afC[0  , 0] := 1.00000E+01; afC[0  , 1] := 1.76331E+00;
afC[1  , 0] := 1.99800E+01; afC[1  , 1] := 1.50760E+00;
afC[2  , 0] := 2.99600E+01; afC[2  , 1] := 1.42075E+00;
afC[3  , 0] := 3.99400E+01; afC[3  , 1] := 1.29546E+00;
afC[4  , 0] := 4.99200E+01; afC[4  , 1] := 1.15214E+00;
afC[5  , 0] := 5.99000E+01; afC[5  , 1] := 1.01763E+00;
afC[6  , 0] := 6.98800E+01; afC[6  , 1] := 9.00494E-01;
afC[7  , 0] := 7.98600E+01; afC[7  , 1] := 8.01146E-01;
afC[8  , 0] := 8.98400E+01; afC[8  , 1] := 7.16659E-01;
afC[9  , 0] := 9.98200E+01; afC[9  , 1] := 6.44674E-01;
afC[10 , 0] := 1.09800E+02; afC[10 , 1] := 5.83258E-01;
afC[11 , 0] := 1.19780E+02; afC[11 , 1] := 5.30612E-01;
afC[12 , 0] := 1.29760E+02; afC[12 , 1] := 4.82622E-01;
afC[13 , 0] := 1.39740E+02; afC[13 , 1] := 4.41233E-01;
afC[14 , 0] := 1.49720E+02; afC[14 , 1] := 4.05363E-01;
afC[15 , 0] := 1.59700E+02; afC[15 , 1] := 3.74061E-01;
afC[16 , 0] := 1.69680E+02; afC[16 , 1] := 3.46568E-01;
afC[17 , 0] := 1.79660E+02; afC[17 , 1] := 3.22281E-01;
afC[18 , 0] := 1.89640E+02; afC[18 , 1] := 3.00702E-01;
afC[19 , 0] := 1.99620E+02; afC[19 , 1] := 2.81430E-01;
afC[20 , 0] := 2.09600E+02; afC[20 , 1] := 2.64143E-01;
afC[21 , 0] := 2.19580E+02; afC[21 , 1] := 2.49090E-01;
afC[22 , 0] := 2.29560E+02; afC[22 , 1] := 2.35204E-01;
afC[23 , 0] := 2.39540E+02; afC[23 , 1] := 2.22562E-01;
afC[24 , 0] := 2.49520E+02; afC[24 , 1] := 2.11150E-01;
afC[25 , 0] := 2.59500E+02; afC[25 , 1] := 2.00952E-01;
afC[26 , 0] := 2.69480E+02; afC[26 , 1] := 1.92300E-01;
afC[27 , 0] := 2.79460E+02; afC[27 , 1] := 1.90036E-01;
afC[28 , 0] := 2.89440E+02; afC[28 , 1] := 3.87092E+00;
afC[29 , 0] := 2.99420E+02; afC[29 , 1] := 3.73978E+00;
afC[30 , 0] := 3.09400E+02; afC[30 , 1] := 3.61374E+00;
afC[31 , 0] := 3.19380E+02; afC[31 , 1] := 3.49365E+00;
afC[32 , 0] := 3.29360E+02; afC[32 , 1] := 3.37555E+00;
afC[33 , 0] := 3.39340E+02; afC[33 , 1] := 3.25992E+00;
afC[34 , 0] := 3.49320E+02; afC[34 , 1] := 3.14769E+00;
afC[35 , 0] := 3.59300E+02; afC[35 , 1] := 3.03887E+00;
afC[36 , 0] := 3.69280E+02; afC[36 , 1] := 2.93349E+00;
afC[37 , 0] := 3.79260E+02; afC[37 , 1] := 2.83161E+00;
afC[38 , 0] := 3.89240E+02; afC[38 , 1] := 2.73380E+00;
afC[39 , 0] := 3.99220E+02; afC[39 , 1] := 2.64002E+00;
afC[40 , 0] := 4.09200E+02; afC[40 , 1] := 2.55009E+00;
afC[41 , 0] := 4.19180E+02; afC[41 , 1] := 2.46405E+00;
afC[42 , 0] := 4.29160E+02; afC[42 , 1] := 2.38175E+00;
afC[43 , 0] := 4.39140E+02; afC[43 , 1] := 2.30302E+00;
afC[44 , 0] := 4.49120E+02; afC[44 , 1] := 2.22778E+00;
afC[45 , 0] := 4.59100E+02; afC[45 , 1] := 2.15582E+00;
afC[46 , 0] := 4.69080E+02; afC[46 , 1] := 2.08703E+00;
afC[47 , 0] := 4.79060E+02; afC[47 , 1] := 2.02128E+00;
afC[48 , 0] := 4.89040E+02; afC[48 , 1] := 1.95840E+00;
afC[49 , 0] := 4.99020E+02; afC[49 , 1] := 1.89825E+00;
afC[50 , 0] := 5.09000E+02; afC[50 , 1] := 1.84069E+00;
afC[51 , 0] := 5.18980E+02; afC[51 , 1] := 1.78566E+00;
afC[52 , 0] := 5.28960E+02; afC[52 , 1] := 1.73294E+00;
afC[53 , 0] := 5.38940E+02; afC[53 , 1] := 1.68243E+00;
afC[54 , 0] := 5.48920E+02; afC[54 , 1] := 1.63403E+00;
afC[55 , 0] := 5.58900E+02; afC[55 , 1] := 1.58768E+00;
afC[56 , 0] := 5.68880E+02; afC[56 , 1] := 1.54316E+00;
afC[57 , 0] := 5.78860E+02; afC[57 , 1] := 1.50047E+00;
afC[58 , 0] := 5.88840E+02; afC[58 , 1] := 1.45950E+00;
afC[59 , 0] := 5.98820E+02; afC[59 , 1] := 1.42015E+00;
afC[60 , 0] := 6.08800E+02; afC[60 , 1] := 1.38232E+00;
afC[61 , 0] := 6.18780E+02; afC[61 , 1] := 1.34605E+00;
afC[62 , 0] := 6.28760E+02; afC[62 , 1] := 1.31107E+00;
afC[63 , 0] := 6.38740E+02; afC[63 , 1] := 1.27742E+00;
afC[64 , 0] := 6.48720E+02; afC[64 , 1] := 1.24507E+00;
afC[65 , 0] := 6.58700E+02; afC[65 , 1] := 1.21392E+00;
afC[66 , 0] := 6.68680E+02; afC[66 , 1] := 1.18394E+00;
afC[67 , 0] := 6.78660E+02; afC[67 , 1] := 1.15506E+00;
afC[68 , 0] := 6.88640E+02; afC[68 , 1] := 1.12719E+00;
afC[69 , 0] := 6.98620E+02; afC[69 , 1] := 1.10028E+00;
afC[70 , 0] := 7.08600E+02; afC[70 , 1] := 1.07436E+00;
afC[71 , 0] := 7.18580E+02; afC[71 , 1] := 1.04930E+00;
afC[72 , 0] := 7.28560E+02; afC[72 , 1] := 1.02513E+00;
afC[73 , 0] := 7.38540E+02; afC[73 , 1] := 1.00175E+00;
afC[74 , 0] := 7.48520E+02; afC[74 , 1] := 9.79159E-01;
afC[75 , 0] := 7.58500E+02; afC[75 , 1] := 9.57327E-01;
afC[76 , 0] := 7.68480E+02; afC[76 , 1] := 9.36210E-01;
afC[77 , 0] := 7.78460E+02; afC[77 , 1] := 9.15783E-01;
afC[78 , 0] := 7.88440E+02; afC[78 , 1] := 8.96007E-01;
afC[79 , 0] := 7.98420E+02; afC[79 , 1] := 8.76865E-01;
afC[80 , 0] := 8.08400E+02; afC[80 , 1] := 8.58327E-01;
afC[81 , 0] := 8.18380E+02; afC[81 , 1] := 8.40363E-01;
afC[82 , 0] := 8.28360E+02; afC[82 , 1] := 8.22948E-01;
afC[83 , 0] := 8.38340E+02; afC[83 , 1] := 8.06071E-01;
afC[84 , 0] := 8.48320E+02; afC[84 , 1] := 7.89702E-01;
afC[85 , 0] := 8.58300E+02; afC[85 , 1] := 7.73825E-01;
afC[86 , 0] := 8.68280E+02; afC[86 , 1] := 7.58419E-01;
afC[87 , 0] := 8.78260E+02; afC[87 , 1] := 7.43465E-01;
afC[88 , 0] := 8.88240E+02; afC[88 , 1] := 7.28939E-01;
afC[89 , 0] := 8.98220E+02; afC[89 , 1] := 7.14835E-01;
afC[90 , 0] := 9.08200E+02; afC[90 , 1] := 7.01136E-01;
afC[91 , 0] := 9.18180E+02; afC[91 , 1] := 6.87817E-01;
afC[92 , 0] := 9.28160E+02; afC[92 , 1] := 6.74868E-01;
afC[93 , 0] := 9.38140E+02; afC[93 , 1] := 6.62286E-01;
afC[94 , 0] := 9.48120E+02; afC[94 , 1] := 6.50047E-01;
afC[95 , 0] := 9.58100E+02; afC[95 , 1] := 6.38137E-01;
afC[96 , 0] := 9.68080E+02; afC[96 , 1] := 6.26556E-01;
afC[97 , 0] := 9.78060E+02; afC[97 , 1] := 6.15276E-01;
afC[98 , 0] := 9.88040E+02; afC[98 , 1] := 6.04299E-01;
afC[99 , 0] := 9.98020E+02; afC[99 , 1] := 5.93605E-01;
afC[100, 0] := 1.00800E+03; afC[100, 1] := 5.83149E-01;
afC[101, 0] := 1.01798E+03; afC[101, 1] := 5.72944E-01;
afC[102, 0] := 1.02796E+03; afC[102, 1] := 5.63003E-01;
afC[103, 0] := 1.03794E+03; afC[103, 1] := 5.53309E-01;
afC[104, 0] := 1.04792E+03; afC[104, 1] := 5.43857E-01;
afC[105, 0] := 1.05790E+03; afC[105, 1] := 5.34649E-01;
afC[106, 0] := 1.06788E+03; afC[106, 1] := 5.25672E-01;
afC[107, 0] := 1.07786E+03; afC[107, 1] := 5.16911E-01;
afC[108, 0] := 1.08784E+03; afC[108, 1] := 5.08374E-01;
afC[109, 0] := 1.09782E+03; afC[109, 1] := 5.00040E-01;
afC[110, 0] := 1.10780E+03; afC[110, 1] := 4.91914E-01;
afC[111, 0] := 1.11778E+03; afC[111, 1] := 4.83987E-01;
afC[112, 0] := 1.12776E+03; afC[112, 1] := 4.76243E-01;
afC[113, 0] := 1.13774E+03; afC[113, 1] := 4.68582E-01;
afC[114, 0] := 1.14772E+03; afC[114, 1] := 4.60764E-01;
afC[115, 0] := 1.15770E+03; afC[115, 1] := 4.53142E-01;
afC[116, 0] := 1.16768E+03; afC[116, 1] := 4.45714E-01;
afC[117, 0] := 1.17766E+03; afC[117, 1] := 4.38467E-01;
afC[118, 0] := 1.18764E+03; afC[118, 1] := 4.31397E-01;
afC[119, 0] := 1.19762E+03; afC[119, 1] := 4.24497E-01;
afC[120, 0] := 1.20760E+03; afC[120, 1] := 4.17760E-01;
afC[121, 0] := 1.21758E+03; afC[121, 1] := 4.11188E-01;
afC[122, 0] := 1.22756E+03; afC[122, 1] := 4.04779E-01;
afC[123, 0] := 1.23754E+03; afC[123, 1] := 3.98516E-01;
afC[124, 0] := 1.24752E+03; afC[124, 1] := 3.92394E-01;
afC[125, 0] := 1.25750E+03; afC[125, 1] := 3.86415E-01;
afC[126, 0] := 1.26748E+03; afC[126, 1] := 3.80576E-01;
afC[127, 0] := 1.27746E+03; afC[127, 1] := 3.74871E-01;
afC[128, 0] := 1.28744E+03; afC[128, 1] := 3.69290E-01;
afC[129, 0] := 1.29742E+03; afC[129, 1] := 3.63839E-01;
afC[130, 0] := 1.30740E+03; afC[130, 1] := 3.58513E-01;
afC[131, 0] := 1.31738E+03; afC[131, 1] := 3.53298E-01;
afC[132, 0] := 1.32736E+03; afC[132, 1] := 3.48197E-01;
afC[133, 0] := 1.33734E+03; afC[133, 1] := 3.43209E-01;
afC[134, 0] := 1.34732E+03; afC[134, 1] := 3.38328E-01;
afC[135, 0] := 1.35730E+03; afC[135, 1] := 3.33549E-01;
afC[136, 0] := 1.36728E+03; afC[136, 1] := 3.28877E-01;
afC[137, 0] := 1.37726E+03; afC[137, 1] := 3.24305E-01;
afC[138, 0] := 1.38724E+03; afC[138, 1] := 3.19827E-01;
afC[139, 0] := 1.39722E+03; afC[139, 1] := 3.15438E-01;
afC[140, 0] := 1.40720E+03; afC[140, 1] := 3.11142E-01;
afC[141, 0] := 1.41718E+03; afC[141, 1] := 3.06937E-01;
afC[142, 0] := 1.42716E+03; afC[142, 1] := 3.02821E-01;
afC[143, 0] := 1.43714E+03; afC[143, 1] := 2.98780E-01;
afC[144, 0] := 1.44712E+03; afC[144, 1] := 2.94825E-01;
afC[145, 0] := 1.45710E+03; afC[145, 1] := 2.90951E-01;
afC[146, 0] := 1.46708E+03; afC[146, 1] := 2.87151E-01;
afC[147, 0] := 1.47706E+03; afC[147, 1] := 2.83423E-01;
afC[148, 0] := 1.48704E+03; afC[148, 1] := 2.79767E-01;
afC[149, 0] := 1.49702E+03; afC[149, 1] := 2.76186E-01;
afC[150, 0] := 1.50700E+03; afC[150, 1] := 2.72675E-01;
afC[151, 0] := 1.51698E+03; afC[151, 1] := 2.69230E-01;
afC[152, 0] := 1.52696E+03; afC[152, 1] := 2.65852E-01;
afC[153, 0] := 1.53694E+03; afC[153, 1] := 2.62539E-01;
afC[154, 0] := 1.54692E+03; afC[154, 1] := 2.59288E-01;
afC[155, 0] := 1.55690E+03; afC[155, 1] := 2.56095E-01;
afC[156, 0] := 1.56688E+03; afC[156, 1] := 2.52961E-01;
afC[157, 0] := 1.57686E+03; afC[157, 1] := 2.49883E-01;
afC[158, 0] := 1.58684E+03; afC[158, 1] := 2.46866E-01;
afC[159, 0] := 1.59682E+03; afC[159, 1] := 2.43905E-01;
afC[160, 0] := 1.60680E+03; afC[160, 1] := 2.40998E-01;
afC[161, 0] := 1.61678E+03; afC[161, 1] := 2.38138E-01;
afC[162, 0] := 1.62676E+03; afC[162, 1] := 2.35331E-01;
afC[163, 0] := 1.63674E+03; afC[163, 1] := 2.32580E-01;
afC[164, 0] := 1.64672E+03; afC[164, 1] := 2.29872E-01;
afC[165, 0] := 1.65670E+03; afC[165, 1] := 2.27208E-01;
afC[166, 0] := 1.66668E+03; afC[166, 1] := 2.24594E-01;
afC[167, 0] := 1.67666E+03; afC[167, 1] := 2.22028E-01;
afC[168, 0] := 1.68664E+03; afC[168, 1] := 2.19509E-01;
afC[169, 0] := 1.69662E+03; afC[169, 1] := 2.17030E-01;
afC[170, 0] := 1.70660E+03; afC[170, 1] := 2.14591E-01;
afC[171, 0] := 1.71658E+03; afC[171, 1] := 2.12193E-01;
afC[172, 0] := 1.72656E+03; afC[172, 1] := 2.09837E-01;
afC[173, 0] := 1.73654E+03; afC[173, 1] := 2.07521E-01;
afC[174, 0] := 1.74652E+03; afC[174, 1] := 2.05243E-01;
afC[175, 0] := 1.75650E+03; afC[175, 1] := 2.03000E-01;
afC[176, 0] := 1.76648E+03; afC[176, 1] := 2.00797E-01;
afC[177, 0] := 1.77646E+03; afC[177, 1] := 1.98631E-01;
afC[178, 0] := 1.78644E+03; afC[178, 1] := 1.96498E-01;
afC[179, 0] := 1.79642E+03; afC[179, 1] := 1.94401E-01;
afC[180, 0] := 1.80640E+03; afC[180, 1] := 1.92342E-01;
afC[181, 0] := 1.81638E+03; afC[181, 1] := 1.90313E-01;
afC[182, 0] := 1.82636E+03; afC[182, 1] := 1.88314E-01;
afC[183, 0] := 1.83634E+03; afC[183, 1] := 1.86346E-01;
afC[184, 0] := 1.84632E+03; afC[184, 1] := 1.84410E-01;
afC[185, 0] := 1.85630E+03; afC[185, 1] := 1.82505E-01;
afC[186, 0] := 1.86628E+03; afC[186, 1] := 1.80630E-01;
afC[187, 0] := 1.87626E+03; afC[187, 1] := 1.78786E-01;
afC[188, 0] := 1.88624E+03; afC[188, 1] := 1.76971E-01;
afC[189, 0] := 1.89622E+03; afC[189, 1] := 1.75181E-01;
afC[190, 0] := 1.90620E+03; afC[190, 1] := 1.73419E-01;
afC[191, 0] := 1.91618E+03; afC[191, 1] := 1.71686E-01;
afC[192, 0] := 1.92616E+03; afC[192, 1] := 1.69979E-01;
afC[193, 0] := 1.93614E+03; afC[193, 1] := 1.68292E-01;
afC[194, 0] := 1.94612E+03; afC[194, 1] := 1.66631E-01;
afC[195, 0] := 1.95610E+03; afC[195, 1] := 1.64998E-01;
afC[196, 0] := 1.96608E+03; afC[196, 1] := 1.63390E-01;
afC[197, 0] := 1.97606E+03; afC[197, 1] := 1.61805E-01;
afC[198, 0] := 1.98604E+03; afC[198, 1] := 1.60243E-01;
afC[199, 0] := 1.99602E+03; afC[199, 1] := 1.58705E-01;
afC[200, 0] := 2.00600E+03; afC[200, 1] := 1.57187E-01;
afC[201, 0] := 2.01598E+03; afC[201, 1] := 1.55689E-01;
afC[202, 0] := 2.02596E+03; afC[202, 1] := 1.54215E-01;
afC[203, 0] := 2.03594E+03; afC[203, 1] := 1.52766E-01;
afC[204, 0] := 2.04592E+03; afC[204, 1] := 1.51337E-01;
afC[205, 0] := 2.05590E+03; afC[205, 1] := 1.49926E-01;
afC[206, 0] := 2.06588E+03; afC[206, 1] := 1.48534E-01;
afC[207, 0] := 2.07586E+03; afC[207, 1] := 1.47161E-01;
afC[208, 0] := 2.08584E+03; afC[208, 1] := 1.45807E-01;
afC[209, 0] := 2.09582E+03; afC[209, 1] := 1.44474E-01;
afC[210, 0] := 2.10580E+03; afC[210, 1] := 1.43160E-01;
afC[211, 0] := 2.11578E+03; afC[211, 1] := 1.41862E-01;
afC[212, 0] := 2.12576E+03; afC[212, 1] := 1.40583E-01;
afC[213, 0] := 2.13574E+03; afC[213, 1] := 1.39320E-01;
afC[214, 0] := 2.14572E+03; afC[214, 1] := 1.38074E-01;
afC[215, 0] := 2.15570E+03; afC[215, 1] := 1.36845E-01;
afC[216, 0] := 2.16568E+03; afC[216, 1] := 1.35632E-01;
afC[217, 0] := 2.17566E+03; afC[217, 1] := 1.34436E-01;
afC[218, 0] := 2.18564E+03; afC[218, 1] := 1.33256E-01;
afC[219, 0] := 2.19562E+03; afC[219, 1] := 1.32091E-01;
afC[220, 0] := 2.20560E+03; afC[220, 1] := 1.30943E-01;
afC[221, 0] := 2.21558E+03; afC[221, 1] := 1.29809E-01;
afC[222, 0] := 2.22556E+03; afC[222, 1] := 1.28692E-01;
afC[223, 0] := 2.23554E+03; afC[223, 1] := 1.27588E-01;
afC[224, 0] := 2.24552E+03; afC[224, 1] := 1.26496E-01;
afC[225, 0] := 2.25550E+03; afC[225, 1] := 1.25418E-01;
afC[226, 0] := 2.26548E+03; afC[226, 1] := 1.24360E-01;
afC[227, 0] := 2.27546E+03; afC[227, 1] := 1.23315E-01;
afC[228, 0] := 2.28544E+03; afC[228, 1] := 1.22280E-01;
afC[229, 0] := 2.29542E+03; afC[229, 1] := 1.21256E-01;
afC[230, 0] := 2.30540E+03; afC[230, 1] := 1.20245E-01;
afC[231, 0] := 2.31538E+03; afC[231, 1] := 1.19249E-01;
afC[232, 0] := 2.32536E+03; afC[232, 1] := 1.18265E-01;
afC[233, 0] := 2.33534E+03; afC[233, 1] := 1.17296E-01;
afC[234, 0] := 2.34532E+03; afC[234, 1] := 1.16340E-01;
afC[235, 0] := 2.35530E+03; afC[235, 1] := 1.15391E-01;
afC[236, 0] := 2.36528E+03; afC[236, 1] := 1.14452E-01;
afC[237, 0] := 2.37526E+03; afC[237, 1] := 1.13527E-01;
afC[238, 0] := 2.38524E+03; afC[238, 1] := 1.12614E-01;
afC[239, 0] := 2.39522E+03; afC[239, 1] := 1.11713E-01;
afC[240, 0] := 2.40520E+03; afC[240, 1] := 1.10822E-01;
afC[241, 0] := 2.41518E+03; afC[241, 1] := 1.09942E-01;
afC[242, 0] := 2.42516E+03; afC[242, 1] := 1.09073E-01;
afC[243, 0] := 2.43514E+03; afC[243, 1] := 1.08214E-01;
afC[244, 0] := 2.44512E+03; afC[244, 1] := 1.07365E-01;
afC[245, 0] := 2.45510E+03; afC[245, 1] := 1.06527E-01;
afC[246, 0] := 2.46508E+03; afC[246, 1] := 1.05698E-01;
afC[247, 0] := 2.47506E+03; afC[247, 1] := 1.04879E-01;
afC[248, 0] := 2.48504E+03; afC[248, 1] := 1.04071E-01;
afC[249, 0] := 2.49502E+03; afC[249, 1] := 1.03272E-01;
afC[250, 0] := 2.50500E+03; afC[250, 1] := 1.02482E-01;
afC[251, 0] := 2.51498E+03; afC[251, 1] := 1.01702E-01;
afC[252, 0] := 2.52496E+03; afC[252, 1] := 1.00928E-01;
afC[253, 0] := 2.53494E+03; afC[253, 1] := 1.00163E-01;
afC[254, 0] := 2.54492E+03; afC[254, 1] := 9.94062E-02;
afC[255, 0] := 2.55490E+03; afC[255, 1] := 9.86599E-02;
afC[256, 0] := 2.56488E+03; afC[256, 1] := 9.79221E-02;
afC[257, 0] := 2.57486E+03; afC[257, 1] := 9.71926E-02;
afC[258, 0] := 2.58484E+03; afC[258, 1] := 9.64715E-02;
afC[259, 0] := 2.59482E+03; afC[259, 1] := 9.57584E-02;
afC[260, 0] := 2.60480E+03; afC[260, 1] := 9.50532E-02;
afC[261, 0] := 2.61478E+03; afC[261, 1] := 9.43559E-02;
afC[262, 0] := 2.62476E+03; afC[262, 1] := 9.36664E-02;
afC[263, 0] := 2.63474E+03; afC[263, 1] := 9.29846E-02;
afC[264, 0] := 2.64472E+03; afC[264, 1] := 9.23104E-02;
afC[265, 0] := 2.65470E+03; afC[265, 1] := 9.16432E-02;
afC[266, 0] := 2.66468E+03; afC[266, 1] := 9.09833E-02;
afC[267, 0] := 2.67466E+03; afC[267, 1] := 9.03306E-02;
afC[268, 0] := 2.68464E+03; afC[268, 1] := 8.96849E-02;
afC[269, 0] := 2.69462E+03; afC[269, 1] := 8.90462E-02;
afC[270, 0] := 2.70460E+03; afC[270, 1] := 8.84147E-02;
afC[271, 0] := 2.71458E+03; afC[271, 1] := 8.77902E-02;
afC[272, 0] := 2.72456E+03; afC[272, 1] := 8.71723E-02;
afC[273, 0] := 2.73454E+03; afC[273, 1] := 8.65608E-02;
afC[274, 0] := 2.74452E+03; afC[274, 1] := 8.59557E-02;
afC[275, 0] := 2.75450E+03; afC[275, 1] := 8.53569E-02;
afC[276, 0] := 2.76448E+03; afC[276, 1] := 8.47644E-02;
afC[277, 0] := 2.77446E+03; afC[277, 1] := 8.41781E-02;
afC[278, 0] := 2.78444E+03; afC[278, 1] := 8.35981E-02;
afC[279, 0] := 2.79442E+03; afC[279, 1] := 8.30244E-02;
afC[280, 0] := 2.80440E+03; afC[280, 1] := 8.24567E-02;
afC[281, 0] := 2.81438E+03; afC[281, 1] := 8.18946E-02;
afC[282, 0] := 2.82436E+03; afC[282, 1] := 8.13382E-02;
afC[283, 0] := 2.83434E+03; afC[283, 1] := 8.07874E-02;
afC[284, 0] := 2.84432E+03; afC[284, 1] := 8.02425E-02;
afC[285, 0] := 2.85430E+03; afC[285, 1] := 7.97031E-02;
afC[286, 0] := 2.86428E+03; afC[286, 1] := 7.91692E-02;
afC[287, 0] := 2.87426E+03; afC[287, 1] := 7.86410E-02;
afC[288, 0] := 2.88424E+03; afC[288, 1] := 7.81182E-02;
afC[289, 0] := 2.89422E+03; afC[289, 1] := 7.76006E-02;
afC[290, 0] := 2.90420E+03; afC[290, 1] := 7.70877E-02;
afC[291, 0] := 2.91418E+03; afC[291, 1] := 7.65800E-02;
afC[292, 0] := 2.92416E+03; afC[292, 1] := 7.60774E-02;
afC[293, 0] := 2.93414E+03; afC[293, 1] := 7.55801E-02;
afC[294, 0] := 2.94412E+03; afC[294, 1] := 7.50877E-02;
afC[295, 0] := 2.95410E+03; afC[295, 1] := 7.46001E-02;
afC[296, 0] := 2.96408E+03; afC[296, 1] := 7.41172E-02;
afC[297, 0] := 2.97406E+03; afC[297, 1] := 7.36390E-02;
afC[298, 0] := 2.98404E+03; afC[298, 1] := 7.31616E-02;
afC[299, 0] := 2.99402E+03; afC[299, 1] := 7.26796E-02;
afC[300, 0] := 3.00400E+03; afC[300, 1] := 7.22023E-02;
afC[301, 0] := 3.01398E+03; afC[301, 1] := 7.17227E-02;
afC[302, 0] := 3.02396E+03; afC[302, 1] := 7.12320E-02;
afC[303, 0] := 3.03394E+03; afC[303, 1] := 7.07462E-02;
afC[304, 0] := 3.04392E+03; afC[304, 1] := 7.02654E-02;
afC[305, 0] := 3.05390E+03; afC[305, 1] := 6.97897E-02;
afC[306, 0] := 3.06388E+03; afC[306, 1] := 6.93187E-02;
afC[307, 0] := 3.07386E+03; afC[307, 1] := 6.88524E-02;
afC[308, 0] := 3.08384E+03; afC[308, 1] := 6.83906E-02;
afC[309, 0] := 3.09382E+03; afC[309, 1] := 6.79334E-02;
afC[310, 0] := 3.10380E+03; afC[310, 1] := 6.74808E-02;
afC[311, 0] := 3.11378E+03; afC[311, 1] := 6.70329E-02;
afC[312, 0] := 3.12376E+03; afC[312, 1] := 6.65895E-02;
afC[313, 0] := 3.13374E+03; afC[313, 1] := 6.61503E-02;
afC[314, 0] := 3.14372E+03; afC[314, 1] := 6.57151E-02;
afC[315, 0] := 3.15370E+03; afC[315, 1] := 6.52841E-02;
afC[316, 0] := 3.16368E+03; afC[316, 1] := 6.48572E-02;
afC[317, 0] := 3.17366E+03; afC[317, 1] := 6.44346E-02;
afC[318, 0] := 3.18364E+03; afC[318, 1] := 6.40161E-02;
afC[319, 0] := 3.19362E+03; afC[319, 1] := 6.36016E-02;
afC[320, 0] := 3.20360E+03; afC[320, 1] := 6.31910E-02;
afC[321, 0] := 3.21358E+03; afC[321, 1] := 6.27843E-02;
afC[322, 0] := 3.22356E+03; afC[322, 1] := 6.23815E-02;
afC[323, 0] := 3.23354E+03; afC[323, 1] := 6.19824E-02;
afC[324, 0] := 3.24352E+03; afC[324, 1] := 6.15871E-02;
afC[325, 0] := 3.25350E+03; afC[325, 1] := 6.11954E-02;
afC[326, 0] := 3.26348E+03; afC[326, 1] := 6.08075E-02;
afC[327, 0] := 3.27346E+03; afC[327, 1] := 6.04235E-02;
afC[328, 0] := 3.28344E+03; afC[328, 1] := 6.00430E-02;
afC[329, 0] := 3.29342E+03; afC[329, 1] := 5.96661E-02;
afC[330, 0] := 3.30340E+03; afC[330, 1] := 5.92926E-02;
afC[331, 0] := 3.31338E+03; afC[331, 1] := 5.89225E-02;
afC[332, 0] := 3.32336E+03; afC[332, 1] := 5.85558E-02;
afC[333, 0] := 3.33334E+03; afC[333, 1] := 5.81925E-02;
afC[334, 0] := 3.34332E+03; afC[334, 1] := 5.78325E-02;
afC[335, 0] := 3.35330E+03; afC[335, 1] := 5.74758E-02;
afC[336, 0] := 3.36328E+03; afC[336, 1] := 5.71223E-02;
afC[337, 0] := 3.37326E+03; afC[337, 1] := 5.67720E-02;
afC[338, 0] := 3.38324E+03; afC[338, 1] := 5.64248E-02;
afC[339, 0] := 3.39322E+03; afC[339, 1] := 5.60808E-02;
afC[340, 0] := 3.40320E+03; afC[340, 1] := 5.57402E-02;
afC[341, 0] := 3.41318E+03; afC[341, 1] := 5.54026E-02;
afC[342, 0] := 3.42316E+03; afC[342, 1] := 5.50681E-02;
afC[343, 0] := 3.43314E+03; afC[343, 1] := 5.47363E-02;
afC[344, 0] := 3.44312E+03; afC[344, 1] := 5.44072E-02;
afC[345, 0] := 3.45310E+03; afC[345, 1] := 5.40811E-02;
afC[346, 0] := 3.46308E+03; afC[346, 1] := 5.37580E-02;
afC[347, 0] := 3.47306E+03; afC[347, 1] := 5.34379E-02;
afC[348, 0] := 3.48304E+03; afC[348, 1] := 5.31207E-02;
afC[349, 0] := 3.49302E+03; afC[349, 1] := 5.28062E-02;
afC[350, 0] := 3.50300E+03; afC[350, 1] := 5.24944E-02;
afC[351, 0] := 3.51298E+03; afC[351, 1] := 5.21853E-02;
afC[352, 0] := 3.52296E+03; afC[352, 1] := 5.18788E-02;
afC[353, 0] := 3.53294E+03; afC[353, 1] := 5.15750E-02;
afC[354, 0] := 3.54292E+03; afC[354, 1] := 5.12739E-02;
afC[355, 0] := 3.55290E+03; afC[355, 1] := 5.09753E-02;
afC[356, 0] := 3.56288E+03; afC[356, 1] := 5.06793E-02;
afC[357, 0] := 3.57286E+03; afC[357, 1] := 5.03859E-02;
afC[358, 0] := 3.58284E+03; afC[358, 1] := 5.00951E-02;
afC[359, 0] := 3.59282E+03; afC[359, 1] := 4.98067E-02;
afC[360, 0] := 3.60280E+03; afC[360, 1] := 4.95208E-02;
afC[361, 0] := 3.61278E+03; afC[361, 1] := 4.92373E-02;
afC[362, 0] := 3.62276E+03; afC[362, 1] := 4.89562E-02;
afC[363, 0] := 3.63274E+03; afC[363, 1] := 4.86774E-02;
afC[364, 0] := 3.64272E+03; afC[364, 1] := 4.84011E-02;
afC[365, 0] := 3.65270E+03; afC[365, 1] := 4.81271E-02;
afC[366, 0] := 3.66268E+03; afC[366, 1] := 4.78554E-02;
afC[367, 0] := 3.67266E+03; afC[367, 1] := 4.75859E-02;
afC[368, 0] := 3.68264E+03; afC[368, 1] := 4.73187E-02;
afC[369, 0] := 3.69262E+03; afC[369, 1] := 4.70536E-02;
afC[370, 0] := 3.70260E+03; afC[370, 1] := 4.67908E-02;
afC[371, 0] := 3.71258E+03; afC[371, 1] := 4.65301E-02;
afC[372, 0] := 3.72256E+03; afC[372, 1] := 4.62716E-02;
afC[373, 0] := 3.73254E+03; afC[373, 1] := 4.60152E-02;
afC[374, 0] := 3.74252E+03; afC[374, 1] := 4.57609E-02;
afC[375, 0] := 3.75250E+03; afC[375, 1] := 4.55086E-02;
afC[376, 0] := 3.76248E+03; afC[376, 1] := 4.52583E-02;
afC[377, 0] := 3.77246E+03; afC[377, 1] := 4.50101E-02;
afC[378, 0] := 3.78244E+03; afC[378, 1] := 4.47639E-02;
afC[379, 0] := 3.79242E+03; afC[379, 1] := 4.45196E-02;
afC[380, 0] := 3.80240E+03; afC[380, 1] := 4.42773E-02;
afC[381, 0] := 3.81238E+03; afC[381, 1] := 4.40370E-02;
afC[382, 0] := 3.82236E+03; afC[382, 1] := 4.37986E-02;
afC[383, 0] := 3.83234E+03; afC[383, 1] := 4.35624E-02;
afC[384, 0] := 3.84232E+03; afC[384, 1] := 4.33281E-02;
afC[385, 0] := 3.85230E+03; afC[385, 1] := 4.30957E-02;
afC[386, 0] := 3.86228E+03; afC[386, 1] := 4.28651E-02;
afC[387, 0] := 3.87226E+03; afC[387, 1] := 4.26360E-02;
afC[388, 0] := 3.88224E+03; afC[388, 1] := 4.24087E-02;
afC[389, 0] := 3.89222E+03; afC[389, 1] := 4.21833E-02;
afC[390, 0] := 3.90220E+03; afC[390, 1] := 4.19596E-02;
afC[391, 0] := 3.91218E+03; afC[391, 1] := 4.17376E-02;
afC[392, 0] := 3.92216E+03; afC[392, 1] := 4.15174E-02;
afC[393, 0] := 3.93214E+03; afC[393, 1] := 4.12989E-02;
afC[394, 0] := 3.94212E+03; afC[394, 1] := 4.10822E-02;
afC[395, 0] := 3.95210E+03; afC[395, 1] := 4.08672E-02;
afC[396, 0] := 3.96208E+03; afC[396, 1] := 4.06539E-02;
afC[397, 0] := 3.97206E+03; afC[397, 1] := 4.04422E-02;
afC[398, 0] := 3.98204E+03; afC[398, 1] := 4.02321E-02;
afC[399, 0] := 3.99202E+03; afC[399, 1] := 4.00236E-02;
afC[400, 0] := 4.00200E+03; afC[400, 1] := 3.98167E-02;
afC[401, 0] := 4.01198E+03; afC[401, 1] := 3.96114E-02;
afC[402, 0] := 4.02196E+03; afC[402, 1] := 3.94077E-02;
afC[403, 0] := 4.03194E+03; afC[403, 1] := 3.92055E-02;
afC[404, 0] := 4.04192E+03; afC[404, 1] := 3.90049E-02;
afC[405, 0] := 4.05190E+03; afC[405, 1] := 3.88058E-02;
afC[406, 0] := 4.06188E+03; afC[406, 1] := 3.86082E-02;
afC[407, 0] := 4.07186E+03; afC[407, 1] := 3.84119E-02;
afC[408, 0] := 4.08184E+03; afC[408, 1] := 3.82172E-02;
afC[409, 0] := 4.09182E+03; afC[409, 1] := 3.80239E-02;
afC[410, 0] := 4.10180E+03; afC[410, 1] := 3.78321E-02;
afC[411, 0] := 4.11178E+03; afC[411, 1] := 3.76418E-02;
afC[412, 0] := 4.12176E+03; afC[412, 1] := 3.74530E-02;
afC[413, 0] := 4.13174E+03; afC[413, 1] := 3.72656E-02;
afC[414, 0] := 4.14172E+03; afC[414, 1] := 3.70795E-02;
afC[415, 0] := 4.15170E+03; afC[415, 1] := 3.68947E-02;
afC[416, 0] := 4.16168E+03; afC[416, 1] := 3.67112E-02;
afC[417, 0] := 4.17166E+03; afC[417, 1] := 3.65291E-02;
afC[418, 0] := 4.18164E+03; afC[418, 1] := 3.63483E-02;
afC[419, 0] := 4.19162E+03; afC[419, 1] := 3.61689E-02;
afC[420, 0] := 4.20160E+03; afC[420, 1] := 3.59908E-02;
afC[421, 0] := 4.21158E+03; afC[421, 1] := 3.58141E-02;
afC[422, 0] := 4.22156E+03; afC[422, 1] := 3.56386E-02;
afC[423, 0] := 4.23154E+03; afC[423, 1] := 3.54643E-02;
afC[424, 0] := 4.24152E+03; afC[424, 1] := 3.52914E-02;
afC[425, 0] := 4.25150E+03; afC[425, 1] := 3.51196E-02;
afC[426, 0] := 4.26148E+03; afC[426, 1] := 3.49491E-02;
afC[427, 0] := 4.27146E+03; afC[427, 1] := 3.47798E-02;
afC[428, 0] := 4.28144E+03; afC[428, 1] := 3.46118E-02;
afC[429, 0] := 4.29142E+03; afC[429, 1] := 3.44449E-02;
afC[430, 0] := 4.30140E+03; afC[430, 1] := 3.42793E-02;
afC[431, 0] := 4.31138E+03; afC[431, 1] := 3.41148E-02;
afC[432, 0] := 4.32136E+03; afC[432, 1] := 3.39516E-02;
afC[433, 0] := 4.33134E+03; afC[433, 1] := 3.37896E-02;
afC[434, 0] := 4.34132E+03; afC[434, 1] := 3.36287E-02;
afC[435, 0] := 4.35130E+03; afC[435, 1] := 3.34689E-02;
afC[436, 0] := 4.36128E+03; afC[436, 1] := 3.33099E-02;
afC[437, 0] := 4.37126E+03; afC[437, 1] := 3.31521E-02;
afC[438, 0] := 4.38124E+03; afC[438, 1] := 3.29954E-02;
afC[439, 0] := 4.39122E+03; afC[439, 1] := 3.28397E-02;
afC[440, 0] := 4.40120E+03; afC[440, 1] := 3.26853E-02;
afC[441, 0] := 4.41118E+03; afC[441, 1] := 3.25321E-02;
afC[442, 0] := 4.42116E+03; afC[442, 1] := 3.23799E-02;
afC[443, 0] := 4.43114E+03; afC[443, 1] := 3.22288E-02;
afC[444, 0] := 4.44112E+03; afC[444, 1] := 3.20787E-02;
afC[445, 0] := 4.45110E+03; afC[445, 1] := 3.19297E-02;
afC[446, 0] := 4.46108E+03; afC[446, 1] := 3.17817E-02;
afC[447, 0] := 4.47106E+03; afC[447, 1] := 3.16348E-02;
afC[448, 0] := 4.48104E+03; afC[448, 1] := 3.14888E-02;
afC[449, 0] := 4.49102E+03; afC[449, 1] := 3.13436E-02;
afC[450, 0] := 4.50100E+03; afC[450, 1] := 3.11994E-02;
afC[451, 0] := 4.51098E+03; afC[451, 1] := 3.10561E-02;
afC[452, 0] := 4.52096E+03; afC[452, 1] := 3.09137E-02;
afC[453, 0] := 4.53094E+03; afC[453, 1] := 3.07725E-02;
afC[454, 0] := 4.54092E+03; afC[454, 1] := 3.06325E-02;
afC[455, 0] := 4.55090E+03; afC[455, 1] := 3.04935E-02;
afC[456, 0] := 4.56088E+03; afC[456, 1] := 3.03553E-02;
afC[457, 0] := 4.57086E+03; afC[457, 1] := 3.02181E-02;
afC[458, 0] := 4.58084E+03; afC[458, 1] := 3.00815E-02;
afC[459, 0] := 4.59082E+03; afC[459, 1] := 2.99458E-02;
afC[460, 0] := 4.60080E+03; afC[460, 1] := 2.98109E-02;
afC[461, 0] := 4.61078E+03; afC[461, 1] := 2.96769E-02;
afC[462, 0] := 4.62076E+03; afC[462, 1] := 2.95439E-02;
afC[463, 0] := 4.63074E+03; afC[463, 1] := 2.94120E-02;
afC[464, 0] := 4.64072E+03; afC[464, 1] := 2.92810E-02;
afC[465, 0] := 4.65070E+03; afC[465, 1] := 2.91508E-02;
afC[466, 0] := 4.66068E+03; afC[466, 1] := 2.90215E-02;
afC[467, 0] := 4.67066E+03; afC[467, 1] := 2.88930E-02;
afC[468, 0] := 4.68064E+03; afC[468, 1] := 2.87653E-02;
afC[469, 0] := 4.69062E+03; afC[469, 1] := 2.86384E-02;
afC[470, 0] := 4.70060E+03; afC[470, 1] := 2.85124E-02;
afC[471, 0] := 4.71058E+03; afC[471, 1] := 2.83872E-02;
afC[472, 0] := 4.72056E+03; afC[472, 1] := 2.82628E-02;
afC[473, 0] := 4.73054E+03; afC[473, 1] := 2.81392E-02;
afC[474, 0] := 4.74052E+03; afC[474, 1] := 2.80163E-02;
afC[475, 0] := 4.75050E+03; afC[475, 1] := 2.78943E-02;
afC[476, 0] := 4.76048E+03; afC[476, 1] := 2.77731E-02;
afC[477, 0] := 4.77046E+03; afC[477, 1] := 2.76527E-02;
afC[478, 0] := 4.78044E+03; afC[478, 1] := 2.75330E-02;
afC[479, 0] := 4.79042E+03; afC[479, 1] := 2.74141E-02;
afC[480, 0] := 4.80040E+03; afC[480, 1] := 2.72960E-02;
afC[481, 0] := 4.81038E+03; afC[481, 1] := 2.71785E-02;
afC[482, 0] := 4.82036E+03; afC[482, 1] := 2.70618E-02;
afC[483, 0] := 4.83034E+03; afC[483, 1] := 2.69458E-02;
afC[484, 0] := 4.84032E+03; afC[484, 1] := 2.68305E-02;
afC[485, 0] := 4.85030E+03; afC[485, 1] := 2.67159E-02;
afC[486, 0] := 4.86028E+03; afC[486, 1] := 2.66022E-02;
afC[487, 0] := 4.87026E+03; afC[487, 1] := 2.64892E-02;
afC[488, 0] := 4.88024E+03; afC[488, 1] := 2.63769E-02;
afC[489, 0] := 4.89022E+03; afC[489, 1] := 2.62653E-02;
afC[490, 0] := 4.90020E+03; afC[490, 1] := 2.61545E-02;
afC[491, 0] := 4.91018E+03; afC[491, 1] := 2.60443E-02;
afC[492, 0] := 4.92016E+03; afC[492, 1] := 2.59347E-02;
afC[493, 0] := 4.93014E+03; afC[493, 1] := 2.58259E-02;
afC[494, 0] := 4.94012E+03; afC[494, 1] := 2.57177E-02;
afC[495, 0] := 4.95010E+03; afC[495, 1] := 2.56102E-02;
afC[496, 0] := 4.96008E+03; afC[496, 1] := 2.55034E-02;
afC[497, 0] := 4.97006E+03; afC[497, 1] := 2.53972E-02;
afC[498, 0] := 4.98004E+03; afC[498, 1] := 2.52917E-02;
afC[499, 0] := 4.99002E+03; afC[499, 1] := 2.51869E-02;
afC[500, 0] := 5.00000E+03; afC[500, 1] := 2.50827E-02;
afC[501, 0] := 5.05000E+03; afC[501, 1] := 2.45704E-02;
afC[502, 0] := 5.10000E+03; afC[502, 1] := 2.40730E-02;
afC[503, 0] := 5.15000E+03; afC[503, 1] := 2.35901E-02;
afC[504, 0] := 5.20000E+03; afC[504, 1] := 2.31214E-02;
afC[505, 0] := 5.25000E+03; afC[505, 1] := 2.26673E-02;
afC[506, 0] := 5.30000E+03; afC[506, 1] := 2.22259E-02;
afC[507, 0] := 5.35000E+03; afC[507, 1] := 2.17882E-02;
afC[508, 0] := 5.40000E+03; afC[508, 1] := 2.13564E-02;
afC[509, 0] := 5.45000E+03; afC[509, 1] := 2.09356E-02;
afC[510, 0] := 5.50000E+03; afC[510, 1] := 2.05272E-02;
afC[511, 0] := 5.55000E+03; afC[511, 1] := 2.01302E-02;
afC[512, 0] := 5.60000E+03; afC[512, 1] := 1.97446E-02;
afC[513, 0] := 5.65000E+03; afC[513, 1] := 1.93698E-02;
afC[514, 0] := 5.70000E+03; afC[514, 1] := 1.90048E-02;
afC[515, 0] := 5.75000E+03; afC[515, 1] := 1.86499E-02;
afC[516, 0] := 5.80000E+03; afC[516, 1] := 1.83050E-02;
afC[517, 0] := 5.85000E+03; afC[517, 1] := 1.79691E-02;
afC[518, 0] := 5.90000E+03; afC[518, 1] := 1.76418E-02;
afC[519, 0] := 5.95000E+03; afC[519, 1] := 1.73236E-02;
afC[520, 0] := 6.00000E+03; afC[520, 1] := 1.70139E-02;
afC[521, 0] := 6.05000E+03; afC[521, 1] := 1.67117E-02;
afC[522, 0] := 6.10000E+03; afC[522, 1] := 1.64175E-02;
afC[523, 0] := 6.15000E+03; afC[523, 1] := 1.61304E-02;
afC[524, 0] := 6.20000E+03; afC[524, 1] := 1.58509E-02;
afC[525, 0] := 6.25000E+03; afC[525, 1] := 1.55788E-02;
afC[526, 0] := 6.30000E+03; afC[526, 1] := 1.53136E-02;
afC[527, 0] := 6.35000E+03; afC[527, 1] := 1.50544E-02;
afC[528, 0] := 6.40000E+03; afC[528, 1] := 1.48015E-02;
afC[529, 0] := 6.45000E+03; afC[529, 1] := 1.45549E-02;
afC[530, 0] := 6.50000E+03; afC[530, 1] := 1.43145E-02;
afC[531, 0] := 6.55000E+03; afC[531, 1] := 1.40799E-02;
afC[532, 0] := 6.60000E+03; afC[532, 1] := 1.38506E-02;
afC[533, 0] := 6.65000E+03; afC[533, 1] := 1.36271E-02;
afC[534, 0] := 6.70000E+03; afC[534, 1] := 1.34088E-02;
afC[535, 0] := 6.75000E+03; afC[535, 1] := 1.31956E-02;
afC[536, 0] := 6.80000E+03; afC[536, 1] := 1.29872E-02;
afC[537, 0] := 6.85000E+03; afC[537, 1] := 1.27830E-02;
afC[538, 0] := 6.90000E+03; afC[538, 1] := 1.25837E-02;
afC[539, 0] := 6.95000E+03; afC[539, 1] := 1.23893E-02;
afC[540, 0] := 7.00000E+03; afC[540, 1] := 1.21996E-02;
afC[541, 0] := 7.05000E+03; afC[541, 1] := 1.20137E-02;
afC[542, 0] := 7.10000E+03; afC[542, 1] := 1.18318E-02;
afC[543, 0] := 7.15000E+03; afC[543, 1] := 1.16536E-02;
afC[544, 0] := 7.20000E+03; afC[544, 1] := 1.14797E-02;
afC[545, 0] := 7.25000E+03; afC[545, 1] := 1.13096E-02;
afC[546, 0] := 7.30000E+03; afC[546, 1] := 1.11430E-02;
afC[547, 0] := 7.35000E+03; afC[547, 1] := 1.09806E-02;
afC[548, 0] := 7.40000E+03; afC[548, 1] := 1.08212E-02;
afC[549, 0] := 7.45000E+03; afC[549, 1] := 1.06649E-02;
afC[550, 0] := 7.50000E+03; afC[550, 1] := 1.05119E-02;
afC[551, 0] := 7.55000E+03; afC[551, 1] := 1.03622E-02;
afC[552, 0] := 7.60000E+03; afC[552, 1] := 1.02157E-02;
afC[553, 0] := 7.65000E+03; afC[553, 1] := 1.00723E-02;
afC[554, 0] := 7.70000E+03; afC[554, 1] := 9.93170E-03;
afC[555, 0] := 7.75000E+03; afC[555, 1] := 9.79384E-03;
afC[556, 0] := 7.80000E+03; afC[556, 1] := 9.65888E-03;
afC[557, 0] := 7.85000E+03; afC[557, 1] := 9.52665E-03;
afC[558, 0] := 7.90000E+03; afC[558, 1] := 9.39708E-03;
afC[559, 0] := 7.95000E+03; afC[559, 1] := 9.27001E-03;
afC[560, 0] := 8.00000E+03; afC[560, 1] := 9.14543E-03;
afC[561, 0] := 8.05000E+03; afC[561, 1] := 9.02332E-03;
afC[562, 0] := 8.10000E+03; afC[562, 1] := 8.90356E-03;
afC[563, 0] := 8.15000E+03; afC[563, 1] := 8.78611E-03;
afC[564, 0] := 8.20000E+03; afC[564, 1] := 8.67093E-03;
afC[565, 0] := 8.25000E+03; afC[565, 1] := 8.55793E-03;
afC[566, 0] := 8.30000E+03; afC[566, 1] := 8.44705E-03;
afC[567, 0] := 8.35000E+03; afC[567, 1] := 8.33832E-03;
afC[568, 0] := 8.40000E+03; afC[568, 1] := 8.23162E-03;
afC[569, 0] := 8.45000E+03; afC[569, 1] := 8.12686E-03;
afC[570, 0] := 8.50000E+03; afC[570, 1] := 8.02406E-03;
afC[571, 0] := 8.55000E+03; afC[571, 1] := 7.92318E-03;
afC[572, 0] := 8.60000E+03; afC[572, 1] := 7.82412E-03;
afC[573, 0] := 8.65000E+03; afC[573, 1] := 7.72686E-03;
afC[574, 0] := 8.70000E+03; afC[574, 1] := 7.63138E-03;
afC[575, 0] := 8.75000E+03; afC[575, 1] := 7.53760E-03;
afC[576, 0] := 8.80000E+03; afC[576, 1] := 7.44546E-03;
afC[577, 0] := 8.85000E+03; afC[577, 1] := 7.35477E-03;
afC[578, 0] := 8.90000E+03; afC[578, 1] := 7.26558E-03;
afC[579, 0] := 8.95000E+03; afC[579, 1] := 7.17504E-03;
afC[580, 0] := 9.00000E+03; afC[580, 1] := 7.08565E-03;
afC[581, 0] := 9.05000E+03; afC[581, 1] := 6.99789E-03;
afC[582, 0] := 9.10000E+03; afC[582, 1] := 6.91169E-03;
afC[583, 0] := 9.15000E+03; afC[583, 1] := 6.82703E-03;
afC[584, 0] := 9.20000E+03; afC[584, 1] := 6.74383E-03;
afC[585, 0] := 9.25000E+03; afC[585, 1] := 6.66206E-03;
afC[586, 0] := 9.30000E+03; afC[586, 1] := 6.58175E-03;
afC[587, 0] := 9.35000E+03; afC[587, 1] := 6.50283E-03;
afC[588, 0] := 9.40000E+03; afC[588, 1] := 6.42530E-03;
afC[589, 0] := 9.45000E+03; afC[589, 1] := 6.34910E-03;
afC[590, 0] := 9.50000E+03; afC[590, 1] := 6.27417E-03;
afC[591, 0] := 9.55000E+03; afC[591, 1] := 6.20050E-03;
afC[592, 0] := 9.60000E+03; afC[592, 1] := 6.12807E-03;
afC[593, 0] := 9.65000E+03; afC[593, 1] := 6.05686E-03;
afC[594, 0] := 9.70000E+03; afC[594, 1] := 5.98686E-03;
afC[595, 0] := 9.75000E+03; afC[595, 1] := 5.91802E-03;
afC[596, 0] := 9.80000E+03; afC[596, 1] := 5.85029E-03;
afC[597, 0] := 9.85000E+03; afC[597, 1] := 5.78369E-03;
afC[598, 0] := 9.90000E+03; afC[598, 1] := 5.71821E-03;
afC[599, 0] := 9.95000E+03; afC[599, 1] := 5.65379E-03;
afC[600, 0] := 1.00000E+04; afC[600, 1] := 5.59040E-03;
afC[601, 0] := 1.00500E+04; afC[601, 1] := 5.52802E-03;
afC[602, 0] := 1.01000E+04; afC[602, 1] := 5.46662E-03;
afC[603, 0] := 1.01500E+04; afC[603, 1] := 5.40620E-03;
afC[604, 0] := 1.02000E+04; afC[604, 1] := 5.34677E-03;
afC[605, 0] := 1.02500E+04; afC[605, 1] := 5.28829E-03;
afC[606, 0] := 1.03000E+04; afC[606, 1] := 5.23074E-03;
afC[607, 0] := 1.03500E+04; afC[607, 1] := 5.17409E-03;
afC[608, 0] := 1.04000E+04; afC[608, 1] := 5.11828E-03;
afC[609, 0] := 1.04500E+04; afC[609, 1] := 5.06334E-03;
afC[610, 0] := 1.05000E+04; afC[610, 1] := 5.00927E-03;
afC[611, 0] := 1.05500E+04; afC[611, 1] := 4.95603E-03;
afC[612, 0] := 1.06000E+04; afC[612, 1] := 4.90356E-03;
afC[613, 0] := 1.06500E+04; afC[613, 1] := 4.85190E-03;
afC[614, 0] := 1.07000E+04; afC[614, 1] := 4.80104E-03;
afC[615, 0] := 1.07500E+04; afC[615, 1] := 4.75096E-03;
afC[616, 0] := 1.08000E+04; afC[616, 1] := 4.70163E-03;
afC[617, 0] := 1.08500E+04; afC[617, 1] := 4.65305E-03;
afC[618, 0] := 1.09000E+04; afC[618, 1] := 4.60518E-03;
afC[619, 0] := 1.09500E+04; afC[619, 1] := 4.55801E-03;
afC[620, 0] := 1.10000E+04; afC[620, 1] := 4.51154E-03;
afC[621, 0] := 1.10500E+04; afC[621, 1] := 4.46577E-03;
afC[622, 0] := 1.11000E+04; afC[622, 1] := 4.42065E-03;
afC[623, 0] := 1.11500E+04; afC[623, 1] := 4.37614E-03;
afC[624, 0] := 1.12000E+04; afC[624, 1] := 4.33228E-03;
afC[625, 0] := 1.12500E+04; afC[625, 1] := 4.28910E-03;
afC[626, 0] := 1.13000E+04; afC[626, 1] := 4.24655E-03;
afC[627, 0] := 1.13500E+04; afC[627, 1] := 4.20459E-03;
afC[628, 0] := 1.14000E+04; afC[628, 1] := 4.16323E-03;
afC[629, 0] := 1.14500E+04; afC[629, 1] := 4.12243E-03;
afC[630, 0] := 1.15000E+04; afC[630, 1] := 4.08220E-03;
afC[631, 0] := 1.15500E+04; afC[631, 1] := 4.04253E-03;
afC[632, 0] := 1.16000E+04; afC[632, 1] := 4.00345E-03;
afC[633, 0] := 1.16500E+04; afC[633, 1] := 3.96490E-03;
afC[634, 0] := 1.17000E+04; afC[634, 1] := 3.92690E-03;
afC[635, 0] := 1.17500E+04; afC[635, 1] := 3.88942E-03;
afC[636, 0] := 1.18000E+04; afC[636, 1] := 3.85244E-03;
afC[637, 0] := 1.18500E+04; afC[637, 1] := 3.81597E-03;
afC[638, 0] := 1.19000E+04; afC[638, 1] := 3.77999E-03;
afC[639, 0] := 1.19500E+04; afC[639, 1] := 3.74450E-03;
afC[640, 0] := 1.20000E+04; afC[640, 1] := 3.70948E-03;
afC[641, 0] := 1.20500E+04; afC[641, 1] := 3.67496E-03;
afC[642, 0] := 1.21000E+04; afC[642, 1] := 3.64090E-03;
afC[643, 0] := 1.21500E+04; afC[643, 1] := 3.60729E-03;
afC[644, 0] := 1.22000E+04; afC[644, 1] := 3.57412E-03;
afC[645, 0] := 1.22500E+04; afC[645, 1] := 3.54139E-03;
afC[646, 0] := 1.23000E+04; afC[646, 1] := 3.50906E-03;
afC[647, 0] := 1.23500E+04; afC[647, 1] := 3.47716E-03;
afC[648, 0] := 1.24000E+04; afC[648, 1] := 3.44569E-03;
afC[649, 0] := 1.24500E+04; afC[649, 1] := 3.41464E-03;
afC[650, 0] := 1.25000E+04; afC[650, 1] := 3.38399E-03;
afC[651, 0] := 1.25500E+04; afC[651, 1] := 3.35374E-03;
afC[652, 0] := 1.26000E+04; afC[652, 1] := 3.32387E-03;
afC[653, 0] := 1.26500E+04; afC[653, 1] := 3.29440E-03;
afC[654, 0] := 1.27000E+04; afC[654, 1] := 3.26532E-03;
afC[655, 0] := 1.27500E+04; afC[655, 1] := 3.23660E-03;
afC[656, 0] := 1.28000E+04; afC[656, 1] := 3.20823E-03;
afC[657, 0] := 1.28500E+04; afC[657, 1] := 3.18023E-03;
afC[658, 0] := 1.29000E+04; afC[658, 1] := 3.15255E-03;
afC[659, 0] := 1.29500E+04; afC[659, 1] := 3.12521E-03;
afC[660, 0] := 1.30000E+04; afC[660, 1] := 3.09821E-03;
afC[661, 0] := 1.30500E+04; afC[661, 1] := 3.07156E-03;
afC[662, 0] := 1.31000E+04; afC[662, 1] := 3.04524E-03;
afC[663, 0] := 1.31500E+04; afC[663, 1] := 3.01926E-03;
afC[664, 0] := 1.32000E+04; afC[664, 1] := 2.99362E-03;
afC[665, 0] := 1.32500E+04; afC[665, 1] := 2.96829E-03;
afC[666, 0] := 1.33000E+04; afC[666, 1] := 2.94325E-03;
afC[667, 0] := 1.33500E+04; afC[667, 1] := 2.91850E-03;
afC[668, 0] := 1.34000E+04; afC[668, 1] := 2.89405E-03;
afC[669, 0] := 1.34500E+04; afC[669, 1] := 2.86991E-03;
afC[670, 0] := 1.35000E+04; afC[670, 1] := 2.84607E-03;
afC[671, 0] := 1.35500E+04; afC[671, 1] := 2.82250E-03;
afC[672, 0] := 1.36000E+04; afC[672, 1] := 2.79922E-03;
afC[673, 0] := 1.36500E+04; afC[673, 1] := 2.77621E-03;
afC[674, 0] := 1.37000E+04; afC[674, 1] := 2.75344E-03;
afC[675, 0] := 1.37500E+04; afC[675, 1] := 2.73094E-03;
afC[676, 0] := 1.38000E+04; afC[676, 1] := 2.70870E-03;
afC[677, 0] := 1.38500E+04; afC[677, 1] := 2.68678E-03;
afC[678, 0] := 1.39000E+04; afC[678, 1] := 2.66511E-03;
afC[679, 0] := 1.39500E+04; afC[679, 1] := 2.64369E-03;
afC[680, 0] := 1.40000E+04; afC[680, 1] := 2.62251E-03;
afC[681, 0] := 1.40500E+04; afC[681, 1] := 2.60157E-03;
afC[682, 0] := 1.41000E+04; afC[682, 1] := 2.58086E-03;
afC[683, 0] := 1.41500E+04; afC[683, 1] := 2.56037E-03;
afC[684, 0] := 1.42000E+04; afC[684, 1] := 2.54011E-03;
afC[685, 0] := 1.42500E+04; afC[685, 1] := 2.52011E-03;
afC[686, 0] := 1.43000E+04; afC[686, 1] := 2.50035E-03;
afC[687, 0] := 1.43500E+04; afC[687, 1] := 2.48082E-03;
afC[688, 0] := 1.44000E+04; afC[688, 1] := 2.46147E-03;
afC[689, 0] := 1.44500E+04; afC[689, 1] := 2.44233E-03;
afC[690, 0] := 1.45000E+04; afC[690, 1] := 2.42340E-03;
afC[691, 0] := 1.45500E+04; afC[691, 1] := 2.40470E-03;
afC[692, 0] := 1.46000E+04; afC[692, 1] := 2.38622E-03;
afC[693, 0] := 1.46500E+04; afC[693, 1] := 2.36794E-03;
afC[694, 0] := 1.47000E+04; afC[694, 1] := 2.34987E-03;
afC[695, 0] := 1.47500E+04; afC[695, 1] := 2.33200E-03;
afC[696, 0] := 1.48000E+04; afC[696, 1] := 2.31432E-03;
afC[697, 0] := 1.48500E+04; afC[697, 1] := 2.29682E-03;
afC[698, 0] := 1.49000E+04; afC[698, 1] := 2.27950E-03;
afC[699, 0] := 1.49500E+04; afC[699, 1] := 2.26238E-03;
afC[700, 0] := 1.50000E+04; afC[700, 1] := 2.24546E-03;
afC[701, 0] := 1.50500E+04; afC[701, 1] := 2.22872E-03;
afC[702, 0] := 1.51000E+04; afC[702, 1] := 2.21217E-03;
afC[703, 0] := 1.51500E+04; afC[703, 1] := 2.19578E-03;
afC[704, 0] := 1.52000E+04; afC[704, 1] := 2.17957E-03;
afC[705, 0] := 1.52500E+04; afC[705, 1] := 2.16353E-03;
afC[706, 0] := 1.53000E+04; afC[706, 1] := 2.14764E-03;
afC[707, 0] := 1.53500E+04; afC[707, 1] := 2.13191E-03;
afC[708, 0] := 1.54000E+04; afC[708, 1] := 2.11636E-03;
afC[709, 0] := 1.54500E+04; afC[709, 1] := 2.10101E-03;
afC[710, 0] := 1.55000E+04; afC[710, 1] := 2.08581E-03;
afC[711, 0] := 1.55500E+04; afC[711, 1] := 2.07078E-03;
afC[712, 0] := 1.56000E+04; afC[712, 1] := 2.05586E-03;
afC[713, 0] := 1.56500E+04; afC[713, 1] := 2.04109E-03;
afC[714, 0] := 1.57000E+04; afC[714, 1] := 2.02648E-03;
afC[715, 0] := 1.57500E+04; afC[715, 1] := 2.01204E-03;
afC[716, 0] := 1.58000E+04; afC[716, 1] := 1.99775E-03;
afC[717, 0] := 1.58500E+04; afC[717, 1] := 1.98361E-03;
afC[718, 0] := 1.59000E+04; afC[718, 1] := 1.96961E-03;
afC[719, 0] := 1.59500E+04; afC[719, 1] := 1.95576E-03;
afC[720, 0] := 1.60000E+04; afC[720, 1] := 1.94205E-03;
afC[721, 0] := 1.60500E+04; afC[721, 1] := 1.92846E-03;
afC[722, 0] := 1.61000E+04; afC[722, 1] := 1.91500E-03;
afC[723, 0] := 1.61500E+04; afC[723, 1] := 1.90168E-03;
afC[724, 0] := 1.62000E+04; afC[724, 1] := 1.88849E-03;
afC[725, 0] := 1.62500E+04; afC[725, 1] := 1.87545E-03;
afC[726, 0] := 1.63000E+04; afC[726, 1] := 1.86254E-03;
afC[727, 0] := 1.63500E+04; afC[727, 1] := 1.84975E-03;
afC[728, 0] := 1.64000E+04; afC[728, 1] := 1.83708E-03;
afC[729, 0] := 1.64500E+04; afC[729, 1] := 1.82454E-03;
afC[730, 0] := 1.65000E+04; afC[730, 1] := 1.81212E-03;
afC[731, 0] := 1.65500E+04; afC[731, 1] := 1.79982E-03;
afC[732, 0] := 1.66000E+04; afC[732, 1] := 1.78764E-03;
afC[733, 0] := 1.66500E+04; afC[733, 1] := 1.77558E-03;
afC[734, 0] := 1.67000E+04; afC[734, 1] := 1.76366E-03;
afC[735, 0] := 1.67500E+04; afC[735, 1] := 1.75186E-03;
afC[736, 0] := 1.68000E+04; afC[736, 1] := 1.74018E-03;
afC[737, 0] := 1.68500E+04; afC[737, 1] := 1.72860E-03;
afC[738, 0] := 1.69000E+04; afC[738, 1] := 1.71710E-03;
afC[739, 0] := 1.69500E+04; afC[739, 1] := 1.70570E-03;
afC[740, 0] := 1.70000E+04; afC[740, 1] := 1.69441E-03;
afC[741, 0] := 1.70500E+04; afC[741, 1] := 1.68327E-03;
afC[742, 0] := 1.71000E+04; afC[742, 1] := 1.67224E-03;
afC[743, 0] := 1.71500E+04; afC[743, 1] := 1.66131E-03;
afC[744, 0] := 1.72000E+04; afC[744, 1] := 1.65047E-03;
afC[745, 0] := 1.72500E+04; afC[745, 1] := 1.63972E-03;
afC[746, 0] := 1.73000E+04; afC[746, 1] := 1.62906E-03;
afC[747, 0] := 1.73500E+04; afC[747, 1] := 1.61850E-03;
afC[748, 0] := 1.74000E+04; afC[748, 1] := 1.60807E-03;
afC[749, 0] := 1.74500E+04; afC[749, 1] := 1.59773E-03;
afC[750, 0] := 1.75000E+04; afC[750, 1] := 1.58749E-03;
afC[751, 0] := 1.75500E+04; afC[751, 1] := 1.57733E-03;
afC[752, 0] := 1.76000E+04; afC[752, 1] := 1.56725E-03;
afC[753, 0] := 1.76500E+04; afC[753, 1] := 1.55726E-03;
afC[754, 0] := 1.77000E+04; afC[754, 1] := 1.54737E-03;
afC[755, 0] := 1.77500E+04; afC[755, 1] := 1.53760E-03;
afC[756, 0] := 1.78000E+04; afC[756, 1] := 1.52791E-03;
afC[757, 0] := 1.78500E+04; afC[757, 1] := 1.51832E-03;
afC[758, 0] := 1.79000E+04; afC[758, 1] := 1.50881E-03;
afC[759, 0] := 1.79500E+04; afC[759, 1] := 1.49937E-03;
afC[760, 0] := 1.80000E+04; afC[760, 1] := 1.49002E-03;
afC[761, 0] := 1.80500E+04; afC[761, 1] := 1.48075E-03;
afC[762, 0] := 1.81000E+04; afC[762, 1] := 1.47156E-03;
afC[763, 0] := 1.81500E+04; afC[763, 1] := 1.46244E-03;
afC[764, 0] := 1.82000E+04; afC[764, 1] := 1.45341E-03;
afC[765, 0] := 1.82500E+04; afC[765, 1] := 1.44446E-03;
afC[766, 0] := 1.83000E+04; afC[766, 1] := 1.43561E-03;
afC[767, 0] := 1.83500E+04; afC[767, 1] := 1.42684E-03;
afC[768, 0] := 1.84000E+04; afC[768, 1] := 1.41814E-03;
afC[769, 0] := 1.84500E+04; afC[769, 1] := 1.40950E-03;
afC[770, 0] := 1.85000E+04; afC[770, 1] := 1.40093E-03;
afC[771, 0] := 1.85500E+04; afC[771, 1] := 1.39243E-03;
afC[772, 0] := 1.86000E+04; afC[772, 1] := 1.38400E-03;
afC[773, 0] := 1.86500E+04; afC[773, 1] := 1.37568E-03;
afC[774, 0] := 1.87000E+04; afC[774, 1] := 1.36743E-03;
afC[775, 0] := 1.87500E+04; afC[775, 1] := 1.35925E-03;
afC[776, 0] := 1.88000E+04; afC[776, 1] := 1.35114E-03;
afC[777, 0] := 1.88500E+04; afC[777, 1] := 1.34311E-03;
afC[778, 0] := 1.89000E+04; afC[778, 1] := 1.33514E-03;
afC[779, 0] := 1.89500E+04; afC[779, 1] := 1.32725E-03;
afC[780, 0] := 1.90000E+04; afC[780, 1] := 1.31941E-03;
afC[781, 0] := 1.90500E+04; afC[781, 1] := 1.31163E-03;
afC[782, 0] := 1.91000E+04; afC[782, 1] := 1.30392E-03;
afC[783, 0] := 1.91500E+04; afC[783, 1] := 1.29627E-03;
afC[784, 0] := 1.92000E+04; afC[784, 1] := 1.28868E-03;
afC[785, 0] := 1.92500E+04; afC[785, 1] := 1.28115E-03;
afC[786, 0] := 1.93000E+04; afC[786, 1] := 1.27368E-03;
afC[787, 0] := 1.93500E+04; afC[787, 1] := 1.26627E-03;
afC[788, 0] := 1.94000E+04; afC[788, 1] := 1.25895E-03;
afC[789, 0] := 1.94500E+04; afC[789, 1] := 1.25168E-03;
afC[790, 0] := 1.95000E+04; afC[790, 1] := 1.24447E-03;
afC[791, 0] := 1.95500E+04; afC[791, 1] := 1.23733E-03;
afC[792, 0] := 1.96000E+04; afC[792, 1] := 1.23024E-03;
afC[793, 0] := 1.96500E+04; afC[793, 1] := 1.22321E-03;
afC[794, 0] := 1.97000E+04; afC[794, 1] := 1.21623E-03;
afC[795, 0] := 1.97500E+04; afC[795, 1] := 1.20931E-03;
afC[796, 0] := 1.98000E+04; afC[796, 1] := 1.20245E-03;
afC[797, 0] := 1.98500E+04; afC[797, 1] := 1.19564E-03;
afC[798, 0] := 1.99000E+04; afC[798, 1] := 1.18889E-03;
afC[799, 0] := 1.99500E+04; afC[799, 1] := 1.18220E-03;
afC[800, 0] := 2.00000E+04; afC[800, 1] := 1.17556E-03;
afC[801, 0] := 2.00500E+04; afC[801, 1] := 1.16897E-03;
afC[802, 0] := 2.01000E+04; afC[802, 1] := 1.16244E-03;
afC[803, 0] := 2.01500E+04; afC[803, 1] := 1.15596E-03;
afC[804, 0] := 2.02000E+04; afC[804, 1] := 1.14953E-03;
afC[805, 0] := 2.02500E+04; afC[805, 1] := 1.14316E-03;
afC[806, 0] := 2.03000E+04; afC[806, 1] := 1.13684E-03;
afC[807, 0] := 2.03500E+04; afC[807, 1] := 1.13057E-03;
afC[808, 0] := 2.04000E+04; afC[808, 1] := 1.12436E-03;
afC[809, 0] := 2.04500E+04; afC[809, 1] := 1.11820E-03;
afC[810, 0] := 2.05000E+04; afC[810, 1] := 1.11208E-03;
afC[811, 0] := 2.05500E+04; afC[811, 1] := 1.10601E-03;
afC[812, 0] := 2.06000E+04; afC[812, 1] := 1.09998E-03;
afC[813, 0] := 2.06500E+04; afC[813, 1] := 1.09400E-03;
afC[814, 0] := 2.07000E+04; afC[814, 1] := 1.08806E-03;
afC[815, 0] := 2.07500E+04; afC[815, 1] := 1.08217E-03;
afC[816, 0] := 2.08000E+04; afC[816, 1] := 1.07631E-03;
afC[817, 0] := 2.08500E+04; afC[817, 1] := 1.07050E-03;
afC[818, 0] := 2.09000E+04; afC[818, 1] := 1.06474E-03;
afC[819, 0] := 2.09500E+04; afC[819, 1] := 1.05902E-03;
afC[820, 0] := 2.10000E+04; afC[820, 1] := 1.05336E-03;
afC[821, 0] := 2.10500E+04; afC[821, 1] := 1.04774E-03;
afC[822, 0] := 2.11000E+04; afC[822, 1] := 1.04217E-03;
afC[823, 0] := 2.11500E+04; afC[823, 1] := 1.03664E-03;
afC[824, 0] := 2.12000E+04; afC[824, 1] := 1.03115E-03;
afC[825, 0] := 2.12500E+04; afC[825, 1] := 1.02570E-03;
afC[826, 0] := 2.13000E+04; afC[826, 1] := 1.02029E-03;
afC[827, 0] := 2.13500E+04; afC[827, 1] := 1.01493E-03;
afC[828, 0] := 2.14000E+04; afC[828, 1] := 1.00960E-03;
afC[829, 0] := 2.14500E+04; afC[829, 1] := 1.00432E-03;
afC[830, 0] := 2.15000E+04; afC[830, 1] := 9.99074E-04;
afC[831, 0] := 2.15500E+04; afC[831, 1] := 9.93871E-04;
afC[832, 0] := 2.16000E+04; afC[832, 1] := 9.88706E-04;
afC[833, 0] := 2.16500E+04; afC[833, 1] := 9.83576E-04;
afC[834, 0] := 2.17000E+04; afC[834, 1] := 9.78485E-04;
afC[835, 0] := 2.17500E+04; afC[835, 1] := 9.73432E-04;
afC[836, 0] := 2.18000E+04; afC[836, 1] := 9.68416E-04;
afC[837, 0] := 2.18500E+04; afC[837, 1] := 9.63439E-04;
afC[838, 0] := 2.19000E+04; afC[838, 1] := 9.58499E-04;
afC[839, 0] := 2.19500E+04; afC[839, 1] := 9.53595E-04;
afC[840, 0] := 2.20000E+04; afC[840, 1] := 9.48727E-04;
afC[841, 0] := 2.20500E+04; afC[841, 1] := 9.43895E-04;
afC[842, 0] := 2.21000E+04; afC[842, 1] := 9.39098E-04;
afC[843, 0] := 2.21500E+04; afC[843, 1] := 9.34336E-04;
afC[844, 0] := 2.22000E+04; afC[844, 1] := 9.29609E-04;
afC[845, 0] := 2.22500E+04; afC[845, 1] := 9.24916E-04;
afC[846, 0] := 2.23000E+04; afC[846, 1] := 9.20259E-04;
afC[847, 0] := 2.23500E+04; afC[847, 1] := 9.15636E-04;
afC[848, 0] := 2.24000E+04; afC[848, 1] := 9.11046E-04;
afC[849, 0] := 2.24500E+04; afC[849, 1] := 9.06489E-04;
afC[850, 0] := 2.25000E+04; afC[850, 1] := 9.01964E-04;
afC[851, 0] := 2.25500E+04; afC[851, 1] := 8.97470E-04;
afC[852, 0] := 2.26000E+04; afC[852, 1] := 8.93008E-04;
afC[853, 0] := 2.26500E+04; afC[853, 1] := 8.88578E-04;
afC[854, 0] := 2.27000E+04; afC[854, 1] := 8.84180E-04;
afC[855, 0] := 2.27500E+04; afC[855, 1] := 8.79814E-04;
afC[856, 0] := 2.28000E+04; afC[856, 1] := 8.75480E-04;
afC[857, 0] := 2.28500E+04; afC[857, 1] := 8.71176E-04;
afC[858, 0] := 2.29000E+04; afC[858, 1] := 8.66903E-04;
afC[859, 0] := 2.29500E+04; afC[859, 1] := 8.62661E-04;
afC[860, 0] := 2.30000E+04; afC[860, 1] := 8.58450E-04;
afC[861, 0] := 2.30500E+04; afC[861, 1] := 8.54268E-04;
afC[862, 0] := 2.31000E+04; afC[862, 1] := 8.50115E-04;
afC[863, 0] := 2.31500E+04; afC[863, 1] := 8.45992E-04;
afC[864, 0] := 2.32000E+04; afC[864, 1] := 8.41894E-04;
afC[865, 0] := 2.32500E+04; afC[865, 1] := 8.37826E-04;
afC[866, 0] := 2.33000E+04; afC[866, 1] := 8.33785E-04;
afC[867, 0] := 2.33500E+04; afC[867, 1] := 8.29772E-04;
afC[868, 0] := 2.34000E+04; afC[868, 1] := 8.25789E-04;
afC[869, 0] := 2.34500E+04; afC[869, 1] := 8.21835E-04;
afC[870, 0] := 2.35000E+04; afC[870, 1] := 8.17909E-04;
afC[871, 0] := 2.35500E+04; afC[871, 1] := 8.14009E-04;
afC[872, 0] := 2.36000E+04; afC[872, 1] := 8.10137E-04;
afC[873, 0] := 2.36500E+04; afC[873, 1] := 8.06288E-04;
afC[874, 0] := 2.37000E+04; afC[874, 1] := 8.02465E-04;
afC[875, 0] := 2.37500E+04; afC[875, 1] := 7.98669E-04;
afC[876, 0] := 2.38000E+04; afC[876, 1] := 7.94898E-04;
afC[877, 0] := 2.38500E+04; afC[877, 1] := 7.91152E-04;
afC[878, 0] := 2.39000E+04; afC[878, 1] := 7.87435E-04;
afC[879, 0] := 2.39500E+04; afC[879, 1] := 7.83743E-04;
afC[880, 0] := 2.40000E+04; afC[880, 1] := 7.80077E-04;
afC[881, 0] := 2.40500E+04; afC[881, 1] := 7.76434E-04;
afC[882, 0] := 2.41000E+04; afC[882, 1] := 7.72817E-04;
afC[883, 0] := 2.41500E+04; afC[883, 1] := 7.69222E-04;
afC[884, 0] := 2.42000E+04; afC[884, 1] := 7.65651E-04;
afC[885, 0] := 2.42500E+04; afC[885, 1] := 7.62104E-04;
afC[886, 0] := 2.43000E+04; afC[886, 1] := 7.58581E-04;
afC[887, 0] := 2.43500E+04; afC[887, 1] := 7.55082E-04;
afC[888, 0] := 2.44000E+04; afC[888, 1] := 7.51605E-04;
afC[889, 0] := 2.44500E+04; afC[889, 1] := 7.48152E-04;
afC[890, 0] := 2.45000E+04; afC[890, 1] := 7.44722E-04;
afC[891, 0] := 2.45500E+04; afC[891, 1] := 7.41315E-04;
afC[892, 0] := 2.46000E+04; afC[892, 1] := 7.37930E-04;
afC[893, 0] := 2.46500E+04; afC[893, 1] := 7.34567E-04;
afC[894, 0] := 2.47000E+04; afC[894, 1] := 7.31226E-04;
afC[895, 0] := 2.47500E+04; afC[895, 1] := 7.27907E-04;
afC[896, 0] := 2.48000E+04; afC[896, 1] := 7.24610E-04;
afC[897, 0] := 2.48500E+04; afC[897, 1] := 7.21334E-04;
afC[898, 0] := 2.49000E+04; afC[898, 1] := 7.18079E-04;
afC[899, 0] := 2.49500E+04; afC[899, 1] := 7.14845E-04;
afC[900, 0] := 2.50000E+04; afC[900, 1] := 7.11633E-04;
afC[901, 0] := 2.50500E+04; afC[901, 1] := 7.08441E-04;
afC[902, 0] := 2.51000E+04; afC[902, 1] := 7.05271E-04;
afC[903, 0] := 2.51500E+04; afC[903, 1] := 7.02121E-04;
afC[904, 0] := 2.52000E+04; afC[904, 1] := 6.98992E-04;
afC[905, 0] := 2.52500E+04; afC[905, 1] := 6.95882E-04;
afC[906, 0] := 2.53000E+04; afC[906, 1] := 6.92793E-04;
afC[907, 0] := 2.53500E+04; afC[907, 1] := 6.89723E-04;
afC[908, 0] := 2.54000E+04; afC[908, 1] := 6.86672E-04;
afC[909, 0] := 2.54500E+04; afC[909, 1] := 6.83640E-04;
afC[910, 0] := 2.55000E+04; afC[910, 1] := 6.80628E-04;
afC[911, 0] := 2.55500E+04; afC[911, 1] := 6.77635E-04;
afC[912, 0] := 2.56000E+04; afC[912, 1] := 6.74661E-04;
afC[913, 0] := 2.56500E+04; afC[913, 1] := 6.71708E-04;
afC[914, 0] := 2.57000E+04; afC[914, 1] := 6.68774E-04;
afC[915, 0] := 2.57500E+04; afC[915, 1] := 6.65857E-04;
afC[916, 0] := 2.58000E+04; afC[916, 1] := 6.62960E-04;
afC[917, 0] := 2.58500E+04; afC[917, 1] := 6.60079E-04;
afC[918, 0] := 2.59000E+04; afC[918, 1] := 6.57215E-04;
afC[919, 0] := 2.59500E+04; afC[919, 1] := 6.54370E-04;
afC[920, 0] := 2.60000E+04; afC[920, 1] := 6.51541E-04;
afC[921, 0] := 2.60500E+04; afC[921, 1] := 6.48731E-04;
afC[922, 0] := 2.61000E+04; afC[922, 1] := 6.45938E-04;
afC[923, 0] := 2.61500E+04; afC[923, 1] := 6.43164E-04;
afC[924, 0] := 2.62000E+04; afC[924, 1] := 6.40407E-04;
afC[925, 0] := 2.62500E+04; afC[925, 1] := 6.37666E-04;
afC[926, 0] := 2.63000E+04; afC[926, 1] := 6.34943E-04;
afC[927, 0] := 2.63500E+04; afC[927, 1] := 6.32236E-04;
afC[928, 0] := 2.64000E+04; afC[928, 1] := 6.29545E-04;
afC[929, 0] := 2.64500E+04; afC[929, 1] := 6.26870E-04;
afC[930, 0] := 2.65000E+04; afC[930, 1] := 6.24212E-04;
afC[931, 0] := 2.65500E+04; afC[931, 1] := 6.21570E-04;
afC[932, 0] := 2.66000E+04; afC[932, 1] := 6.18944E-04;
afC[933, 0] := 2.66500E+04; afC[933, 1] := 6.16299E-04;
afC[934, 0] := 2.67000E+04; afC[934, 1] := 6.13659E-04;
afC[935, 0] := 2.67500E+04; afC[935, 1] := 6.11036E-04;
afC[936, 0] := 2.68000E+04; afC[936, 1] := 6.08428E-04;
afC[937, 0] := 2.68500E+04; afC[937, 1] := 6.05837E-04;
afC[938, 0] := 2.69000E+04; afC[938, 1] := 6.03251E-04;
afC[939, 0] := 2.69500E+04; afC[939, 1] := 6.00667E-04;
afC[940, 0] := 2.70000E+04; afC[940, 1] := 5.98099E-04;
afC[941, 0] := 2.70500E+04; afC[941, 1] := 5.95547E-04;
afC[942, 0] := 2.71000E+04; afC[942, 1] := 5.93011E-04;
afC[943, 0] := 2.71500E+04; afC[943, 1] := 5.90490E-04;
afC[944, 0] := 2.72000E+04; afC[944, 1] := 5.87986E-04;
afC[945, 0] := 2.72500E+04; afC[945, 1] := 5.85497E-04;
afC[946, 0] := 2.73000E+04; afC[946, 1] := 5.83023E-04;
afC[947, 0] := 2.73500E+04; afC[947, 1] := 5.80564E-04;
afC[948, 0] := 2.74000E+04; afC[948, 1] := 5.78120E-04;
afC[949, 0] := 2.74500E+04; afC[949, 1] := 5.75690E-04;
afC[950, 0] := 2.75000E+04; afC[950, 1] := 5.73274E-04;
afC[951, 0] := 2.75500E+04; afC[951, 1] := 5.70873E-04;
afC[952, 0] := 2.76000E+04; afC[952, 1] := 5.68486E-04;
afC[953, 0] := 2.76500E+04; afC[953, 1] := 5.66113E-04;
afC[954, 0] := 2.77000E+04; afC[954, 1] := 5.63755E-04;
afC[955, 0] := 2.77500E+04; afC[955, 1] := 5.61409E-04;
afC[956, 0] := 2.78000E+04; afC[956, 1] := 5.59077E-04;
afC[957, 0] := 2.78500E+04; afC[957, 1] := 5.56759E-04;
afC[958, 0] := 2.79000E+04; afC[958, 1] := 5.54454E-04;
afC[959, 0] := 2.79500E+04; afC[959, 1] := 5.52164E-04;
afC[960, 0] := 2.80000E+04; afC[960, 1] := 5.49887E-04;
afC[961, 0] := 2.80500E+04; afC[961, 1] := 5.47625E-04;
afC[962, 0] := 2.81000E+04; afC[962, 1] := 5.45376E-04;
afC[963, 0] := 2.81500E+04; afC[963, 1] := 5.43140E-04;
afC[964, 0] := 2.82000E+04; afC[964, 1] := 5.40918E-04;
afC[965, 0] := 2.82500E+04; afC[965, 1] := 5.38708E-04;
afC[966, 0] := 2.83000E+04; afC[966, 1] := 5.36512E-04;
afC[967, 0] := 2.83500E+04; afC[967, 1] := 5.34329E-04;
afC[968, 0] := 2.84000E+04; afC[968, 1] := 5.32159E-04;
afC[969, 0] := 2.84500E+04; afC[969, 1] := 5.30001E-04;
afC[970, 0] := 2.85000E+04; afC[970, 1] := 5.27856E-04;
afC[971, 0] := 2.85500E+04; afC[971, 1] := 5.25723E-04;
afC[972, 0] := 2.86000E+04; afC[972, 1] := 5.23601E-04;
afC[973, 0] := 2.86500E+04; afC[973, 1] := 5.21492E-04;
afC[974, 0] := 2.87000E+04; afC[974, 1] := 5.19394E-04;
afC[975, 0] := 2.87500E+04; afC[975, 1] := 5.17309E-04;
afC[976, 0] := 2.88000E+04; afC[976, 1] := 5.15235E-04;
afC[977, 0] := 2.88500E+04; afC[977, 1] := 5.13175E-04;
afC[978, 0] := 2.89000E+04; afC[978, 1] := 5.11126E-04;
afC[979, 0] := 2.89500E+04; afC[979, 1] := 5.09090E-04;
afC[980, 0] := 2.90000E+04; afC[980, 1] := 5.07065E-04;
afC[981, 0] := 2.90500E+04; afC[981, 1] := 5.05051E-04;
afC[982, 0] := 2.91000E+04; afC[982, 1] := 5.03049E-04;
afC[983, 0] := 2.91500E+04; afC[983, 1] := 5.01058E-04;
afC[984, 0] := 2.92000E+04; afC[984, 1] := 4.99077E-04;
afC[985, 0] := 2.92500E+04; afC[985, 1] := 4.97108E-04;
afC[986, 0] := 2.93000E+04; afC[986, 1] := 4.95150E-04;
afC[987, 0] := 2.93500E+04; afC[987, 1] := 4.93203E-04;
afC[988, 0] := 2.94000E+04; afC[988, 1] := 4.91267E-04;
afC[989, 0] := 2.94500E+04; afC[989, 1] := 4.89341E-04;
afC[990, 0] := 2.95000E+04; afC[990, 1] := 4.87427E-04;
afC[991, 0] := 2.95500E+04; afC[991, 1] := 4.85523E-04;
afC[992, 0] := 2.96000E+04; afC[992, 1] := 4.83630E-04;
afC[993, 0] := 2.96500E+04; afC[993, 1] := 4.81748E-04;
afC[994, 0] := 2.97000E+04; afC[994, 1] := 4.79875E-04;
afC[995, 0] := 2.97500E+04; afC[995, 1] := 4.78013E-04;
afC[996, 0] := 2.98000E+04; afC[996, 1] := 4.76161E-04;
afC[997, 0] := 2.98500E+04; afC[997, 1] := 4.74319E-04;
afC[998, 0] := 2.99000E+04; afC[998, 1] := 4.72488E-04;
afC[999, 0] := 2.99500E+04; afC[999, 1] := 4.70666E-04;

// Element = Al

